// This function has been automatically generated from the project information.
{attribute 'signature_flag' := '1073741824'}
{attribute 'TcGenerated'}
{attribute 'no-analysis'}
FUNCTION F_GetCompany : WSTRING
VAR_INPUT
	
END_VAR

F_GetCompany := "Beckhoff Automation LLC.";

END_FUNCTION

(* stored: Version 1.1.0.1
   POU F_GetCompany: Id {a23acc66-f809-457f-a3eb-cc17e799ea45}, SpecialFunc None *)
